FUNCTION_BLOCK FB_OrangeConveyor
VAR
	Motor					:FB_ConveyorMotor;
	LTU						:FB_LTU_Cylinder;	
    BlueStopper				:FB_Stopper;
	PurpleStopper_1			:FB_Stopper;
	PurpleStopper_2			:FB_Stopper;
    nStatus					:INT:=0;					
END_VAR

END_FUNCTION_BLOCK

(* stored: Version 1.1.0.1, ProductVersion 3.1.4024.12
   POU FB_OrangeConveyor: Id {2bfa092c-6bf0-4d1c-991c-224c2a5d6655}, SpecialFunc None *)
